# EPICS StreamDevice protocol: devAPPNAME.proto
ReplyTimeout = 500;
OutTerminator = "\r\n";

@writetimeout { disconnect; }
@replytimeout { disconnect; }
@readtimeout  { disconnect; }
@mismatch     { disconnect; }

getIDN {
    out "*IDN?";
    in "%\$1[^\r\n]";
    ExtraInput = Ignore;
}
